FUNCTION_BLOCK WAGOConveyorControllerECC (* Basic HCECC Function Block Type *)
  (* Standard: 61499-2 *)
  (* Version 0.0, 2007-06-26, GDS, University of Auckland *)
  (* Compiler header: package fb.rt.wago; *)
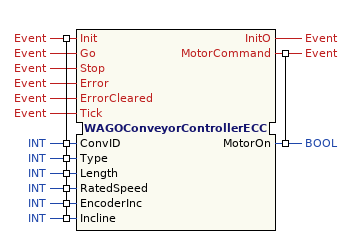
  EVENT_INPUT
    Init WITH ConvID, Type, Length, RatedSpeed, EncoderInc, Incline;
    Go;
    Stop;
    Error;
    ErrorCleared;
    Tick;
  END_EVENT
  EVENT_OUTPUT
    InitO; (* Initialization Confirm *)
    MotorCommand WITH MotorOn;
  END_EVENT
  VAR_INPUT
    ConvID : INT;
    Type : INT;
    Length : INT;
    RatedSpeed : INT;
    EncoderInc : INT;
    Incline : INT;
  END_VAR
  VAR_OUTPUT
    MotorOn : BOOL;
  END_VAR
  VAR
    ResultCode : INT;
    BagsInModel : INT := 0;
  END_VAR
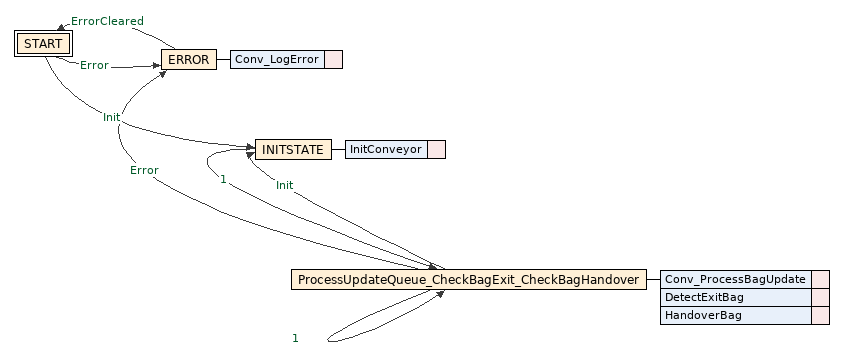
  EC_STATES
    START; (* Initial State *)
    ERROR : Conv_LogError; (* Initialization *)
    INITSTATE : InitConveyor;
    ProcessUpdateQueue_CheckBagExit_CheckBagHandover : Conv_ProcessBagUpdate, DetectExitBag, HandoverBag; (* Cross Product State *)
  END_STATES
  EC_TRANSITIONS
    ERROR TO START := ErrorCleared;
    ProcessUpdateQueue_CheckBagExit_CheckBagHandover TO ERROR := Error;
    START TO ERROR := Error;
    ProcessUpdateQueue_CheckBagExit_CheckBagHandover TO INITSTATE := Init;
    START TO INITSTATE := Init;
    ProcessUpdateQueue_CheckBagExit_CheckBagHandover TO ProcessUpdateQueue_CheckBagExit_CheckBagHandover := 1;
    INITSTATE TO ProcessUpdateQueue_CheckBagExit_CheckBagHandover := 1;
  END_TRANSITIONS
  ALGORITHM Conv_HandleBagDetect IN C:
//TODO: Rename to Conv_ProcessUpdateBag.. no args.... Hmmm
void Conv_HandleBagDetect(int ConvID)
{
 // Loop through all PEs in ConvPtr.PE and Update accordingly
 // vars for search
 int ordHighLimit, ordLowLimit, TrackTolerance;
 // return vars from Conv_SearchModelForBag
 int searchResultCode, ModelPtr = MATCH_NONE, BagFoundDistance;

 // Bag data...
 int BagID;

 // Update Bag Data
 int updateResultCode;
//Conv[ConvID].Slow.PE[6].Detect
// StateLast
// ObjectStartEncCount
// BagDSEncCount
// BagUSEncCount
//AssObjDSEncCount, AssObjUSEncCount
// TODO: ********* NULL
BagUpdateEventRecordStruct UpdateRecord;
// RETURNS from UpdateBag
int LastUpdateBagID, LastObjectTrackStatus;

 int PEID;
 printf("Conv %d detected a bag edge\n", ConvID);
 for (PEID = 0; PEID <6; PEID++) {
   //if PE is configured...
   if( Conv[ConvID].Config.UpdateDev[PEID].Type == UPDATEDEVTYPE_NONE) break; // they will be in order... so no more PEs after this 'non'- PE

    TrackTolerance = Conv[ConvID].Config.UpdateDev[PEID].TrackTolerance;
    // Do it
    if (Conv[ConvID].Slow.PE[PEID].LeadingEdgeEvent == true) {
  printf("*\t\tLeadingEdgeEvent Detected on PE %d\n", PEID);
  // Populate UpdateRecord
  UpdateRecord.ConvID = ConvID;
  UpdateRecord.UpdateDevID = PEID;
  UpdateRecord.BagID = NO_DATA;
  UpdateRecord.BagDSEncCount = Conv[ConvID].Slow.PE[PEID].PEBlockedEncCount;
  UpdateRecord.BagUSEncCount = NO_DATA;
  UpdateRecord.BagUSEncCountOnDSConv = NO_DATA;

  Conv_UpdateBag(UPDATETYPE_DS, UpdateRecord, TrackTolerance, POSITIONDATA_EXPECTED, &updateResultCode, &LastUpdateBagID, &LastObjectTrackStatus);

     // check result code...
     // not yet
     Conv[ConvID].Slow.PE[PEID].LeadingEdgeEvent = false;
  printf("Conv[ConvID].Slow.UpdateDev[PEID].LastUpdateBagID = %d\n", Conv[ConvID].Slow.UpdateDev[PEID].LastUpdateBagID);
    }
    else if (Conv[ConvID].Slow.PE[PEID].TrailingEdgeEvent == true)  {
  printf("*\t\tTrailingEdgeEvent Detected on Conv[%d], PE %d\n", ConvID, PEID);
  // Search model for bag (details)
  /*int BagUSOrdLimit, BagDSOrdLimit;
  BagDSOrdLimit = Conv[ConvID].Slow.PE[PEID].PEUnblockedEncCount - TrackTolerance;
  if( BagDSOrdLimit < 0 )
  {
   BagDSOrdLimit = 0;
  }
  BagUSOrdLimit = Conv[ConvID].Slow.PE[PEID].PEUnblockedEncCount + TrackTolerance;
  Conv_SearchModelForBag(0, ConvID, SEARCHTYPE_US, BagUSOrdLimit, BagDSOrdLimit, &searchResultCode, &ModelPtr, &BagFoundDistance);
  if( ModelPtr == MATCH_NONE )
  {
   printf("Bag Not Found for BagDSOrdLimit %d and BagUSOrdLimit %d\n", BagDSOrdLimit, BagUSOrdLimit);
   Conv[ConvID].Slow.PE[PEID].TrailingEdgeEvent = false;
   continue;
  }*/
  // Populate UpdateRecord
  UpdateRecord.ConvID = ConvID;
  UpdateRecord.UpdateDevID = PEID;
  printf("Conv[ConvID].Slow.UpdateDev[PEID].LastUpdateBagID = %d\n", Conv[ConvID].Slow.UpdateDev[PEID].LastUpdateBagID);
  UpdateRecord.BagID = Conv[ConvID].Slow.UpdateDev[PEID].LastUpdateBagID; //ModelPtr;
  UpdateRecord.BagDSEncCount = NO_DATA;
  UpdateRecord.BagUSEncCount = Conv[ConvID].Slow.PE[PEID].PEUnblockedEncCount;
  //TODO: Should NOT be null
  //The encoder count on the DOWNSTREAM conveyor when the upstream end of a confirmed bag was last detected
  UpdateRecord.BagUSEncCountOnDSConv = NO_DATA;

  Conv_UpdateBag(UPDATETYPE_US, UpdateRecord, TrackTolerance, POSITIONDATA_EXPECTED, &updateResultCode, &LastUpdateBagID, &LastObjectTrackStatus);
  // check result code...

  // not yet
  Conv[ConvID].Slow.PE[PEID].TrailingEdgeEvent = false;
  Conv[ConvID].Slow.UpdateDev[PEID].LastUpdateBagID = Conv[ConvID].Slow.Model.Bag[ModelPtr];
    }
 } // end for

}
  END_ALGORITHM
  ALGORITHM Conv_MotorGo IN C:
void Conv_MotorGo(ConveyorController_HCECC_ECC* me)
{
 me->MotorOn = true;
}
  END_ALGORITHM
  ALGORITHM Conv_MotorStop IN C:
void Conv_MotorStop(ConveyorController_HCECC_ECC* me)
{
 me->MotorOn = false;
}
  END_ALGORITHM
  ALGORITHM InitConveyor IN C:
void InitConveyor(ConveyorController_HCECC_ECC* me)
{
 printf("Conv[%d] InitConv (Empty Function)\n", me->ConvID);
}
  END_ALGORITHM
END_FUNCTION_BLOCK
